(* PLC project SafeLOGIC-1, BrAutomation SafeDESIGNER  4.3.4.4 *)
(* stored: companyURL http://www.br-automation.com, creationDateTime Thu Jun 24 15:44:02 2021 *)

PROGRAM Main
  VAR  (* added by the conversion: wires and edge detectors of the diagram *)
    _SAFEBOOL_TO_BOOL27_OUT : BOOL;
  END_VAR

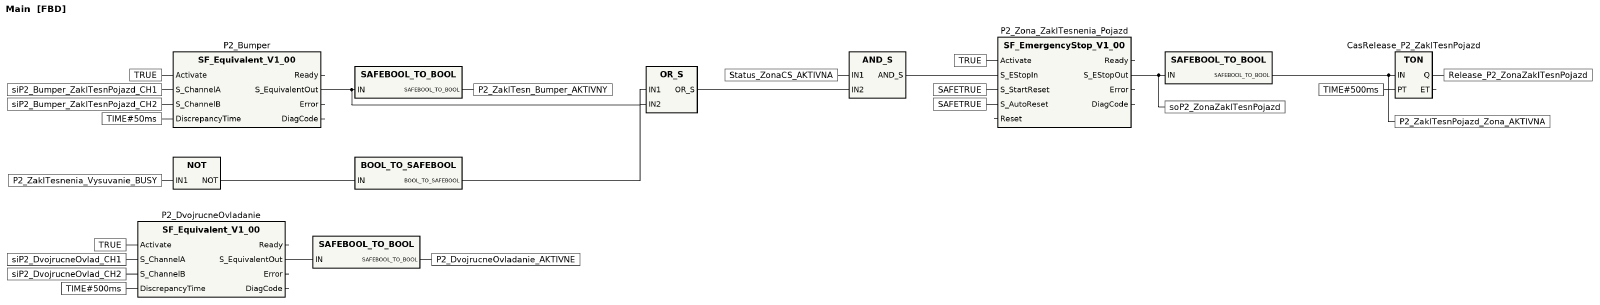
(* FBD diagram, written out as Structured Text *)
P2_Bumper(Activate := TRUE, S_ChannelA := siP2_Bumper_ZaklTesnPojazd_CH1, S_ChannelB := siP2_Bumper_ZaklTesnPojazd_CH2, DiscrepancyTime := TIME#50ms);
P2_Zona_ZaklTesnenia_Pojazd(Activate := TRUE, S_EStopIn := AND_S(Status_ZonaCS_AKTIVNA, OR_S(P2_Bumper.S_EquivalentOut, BOOL_TO_SAFEBOOL(NOT P2_ZaklTesnenia_Vysuvanie_BUSY))), S_StartReset := SAFETRUE, S_AutoReset := SAFETRUE);
soP2_ZonaZaklTesnPojazd := P2_Zona_ZaklTesnenia_Pojazd.S_EStopOut;
_SAFEBOOL_TO_BOOL27_OUT := SAFEBOOL_TO_BOOL(P2_Zona_ZaklTesnenia_Pojazd.S_EStopOut);
P2_ZaklTesnPojazd_Zona_AKTIVNA := _SAFEBOOL_TO_BOOL27_OUT;
CasRelease_P2_ZaklTesnPojazd(IN := _SAFEBOOL_TO_BOOL27_OUT, PT := TIME#500ms);
Release_P2_ZonaZaklTesnPojazd := CasRelease_P2_ZaklTesnPojazd.Q;
P2_ZaklTesn_Bumper_AKTIVNY := SAFEBOOL_TO_BOOL(P2_Bumper.S_EquivalentOut);
P2_DvojrucneOvladanie(Activate := TRUE, S_ChannelA := siP2_DvojrucneOvlad_CH1, S_ChannelB := siP2_DvojrucneOvlad_CH2, DiscrepancyTime := TIME#500ms);
P2_DvojrucneOvladanie_AKTIVNE := SAFEBOOL_TO_BOOL(P2_DvojrucneOvladanie.S_EquivalentOut);
END_PROGRAM
